Staubli VAL3: OnF3.pgx

program OnF3()
begin
  //
  switch nPage
    case 0
      pdemo[nSelected]=here(t2,frmaster)
    break
    case 1

    break
  endSwitch
end
